Staubli VAL3: onStart.pgx

program onStart()
  local num i
  local string l_sMessage
begin
  // wait the START
  wait(cycleStatus:nInterfaceToSV==-1)
  cls()
  //
  setTextMode(0)
  // INIT
  if saveData:mode<2
    userPage(true)
  else
    userPage(false)
  endIf
  //
  logMsg("[KERNEL] INTERFACE:PAGE Home Page, version: " +sVersion)
  //
  // init the session
  // change session
  call language:message(l_sMessage,19)
  l_sMessage=l_sMessage+" SESSION DATA..."
  call use:timerDialog(l_sMessage,0)
  call saveData:changeSession(saveData:sSession)
  call processList:loadProcessList(i)
  // continue
  use:bUseRefresh=true
end
